(* IEC 61131-3 sources: vscode-twincat-st/src/sample/Errors, 25 files *)

(* ---- C0001.st ---- *)
// C0001: Constant '{constant}' too large for type '{name}'
FUNCTION_BLOCK C0001

    VAR

        // Signed Integer Types
        _int1:                  INT             := INT#2#10000000_00000000;
        _int2:                  INT             := INT#16#8000;

        // Unsigned Integer Types
        _uint1:                 UINT            := UINT#-1;
        _Uint2:                 UINT            := 18446744073709551616;

        // Floating Point Types
        _real:                  REAL            := REAL#3.402824E+38;
        _lreal:                 LREAL           := LREAL#1.7976931348623159e+308;
        _lreal2:                LREAL           := 1.7976931348623159e+308;

        // Time-Related Types
        time_over1:             TIME            := TIME#1M61S;
        time_over2:             TIME            := TIME#49D17H2M47S296MS;

        date_under:             DATE            := DATE#1969-12-31;
		date_over:              DATE            := DATE#2106-02-08;
        date_invalid:           DATE            := D#1970-01-40;

        date_and_time_under:    DATE_AND_TIME   := DATE_AND_TIME#1969-12-31-23:59:59;
        date_and_time_over:     DATE_AND_TIME   := DATE_AND_TIME#2106-02-07-06:28:16;
        date_and_time_invalid:  DATE_AND_TIME   := DATE_AND_TIME#1970-01-40-00:00:00;

        time_of_day_over:       TIME_OF_DAY     := TIME_OF_DAY#24:00:00.000;
        time_of_day_invalid:    TIME_OF_DAY     := TIME_OF_DAY#23:00:72.000;

        l_time_over1:           LTIME           := LTIME#1M61S;
        l_time_over2:           LTIME           := LTIME#213503D23H34M33S709MS551US616NS;

        l_date_under:           LDATE           := LDATE#1969-12-31;
		l_date_over:            LDATE           := LDATE#2554-07-22;

        l_date_and_time_under:  LDATE_AND_TIME  := LDATE_AND_TIME#1969-12-31-23:59:59;
        l_date_and_time_over:   LDATE_AND_TIME  := LDATE_AND_TIME#2554-7-21-23:34:33.709551616;

        l_time_of_day_over:     LTIME_OF_DAY    := LTIME_OF_DAY#24:00:00.000;
    END_VAR
END_FUNCTION_BLOCK

(* ---- C0018.st ---- *)
// C0018 '{name}' is no valid assignment target
FUNCTION_BLOCK C0018

    VAR CONSTANT
        _a: INT;
    END_VAR

    PROPERTY A : INT
        GET
            //
        END_GET
    END_PROPERTY

    METHOD B
        //
    END_METHOD

    _a  := 1;
    A   := 1;
    B   := 1;
END_FUNCTION_BLOCK

(* ---- C0032_DUTs.st ---- *)
// C0032: Cannot convert type '{type}' to type '{type}'

TYPE U_C0032 :
UNION
    A: USINT := 1024;
END_UNION
END_TYPE

TYPE ST_C0032 :
STRUCT
    A: USINT := 1024;
END_STRUCT
END_TYPE

TYPE E_C0032_Default :
(
    A
);
END_TYPE

TYPE E_C0032_USINT :
(
    A := 1024
) USINT;
END_TYPE

TYPE C0032_InnerAlias : E_C0032_USINT;
END_TYPE

TYPE C0032_OuterAlias : C0032_InnerAlias;
END_TYPE

FUNCTION_BLOCK C0032_DUTs

    VAR
        _enum_default:      E_C0032_Default     := 32768;
        _enum_usint:        E_C0032_USINT       := 256;
        _alias:             C0032_OuterAlias    := 256;
        _assign_from_x_1:   USINT               := E_C0032_Default.A;
        _assign_from_x_2:   BOOL;
    END_VAR

    _enum_default       := 32768;
    _enum_usint         := 256;
    _alias              := 256;
    _assign_from_x_1    := E_C0032_Default.A;
    _assign_from_x_1    := _enum_default;
    _assign_from_x_2    := _alias;
END_FUNCTION_BLOCK

(* ---- C0032_Literals.st ---- *)
// C0032: Cannot convert type '{type}' to type '{type}'

FUNCTION_BLOCK C0032_Literals

    VAR

        _a:         BOOL        := 2;
        _subrange:  INT(1..1)   := 2;
    END_VAR

    _a          := 2;
    _subrange   := 2;
END_FUNCTION_BLOCK

(* ---- C0032_Variables.st ---- *)
// C0032: Cannot convert type '{type}' to type '{type}'
// https://infosys.beckhoff.com/english.php?content=../content/1033/tf5100_tc3_nc_i/4188351883.html&id=
FUNCTION_BLOCK C0032_Variables

    VAR
        _bool:  BOOL;
        _byte:  BYTE;
    END_VAR

    _bool := _byte;     // Byte
    _bool := -_byte;    // INT
    _bool := -BYTE#1;   // SINT
END_FUNCTION_BLOCK

(* ---- C0035.st ---- *)
// C0035: Program name, function or function block instance expected instead of '{name}'
FUNCTION_BLOCK FB_C0035

    VAR
        _a: INT;
    END_VAR

    PROPERTY A : INT
        GET
            //
        END_GET
    END_PROPERTY

    METHOD M_A : INT
        //
    END_METHOD

    _a();
    _a := _a();
    E_C0035.a();

    _a := A();
    A();
END_FUNCTION_BLOCK

TYPE E_C0035 :
(
    a
);
END_TYPE

(* ---- C0036.st ---- *)
// C0036: Cannot call object of type '{name}'
FUNCTION_BLOCK FB_C0036
    GVL_C0036();
    E_C0036();
    ST_C0036();
    U_C0036();
END_FUNCTION_BLOCK

VAR_GLOBAL GVL_C0036
    //
END_VAR

TYPE E_C0036 :
(
    dummy
);
END_TYPE

TYPE ST_C0036 :
STRUCT
    //
END_STRUCT
END_TYPE

TYPE U_C0036 :
UNION
    //
END_UNION
END_TYPE

(* ---- C0037.st ---- *)
// C0037: '{name}' is no input of '{name}'

FUNCTION_BLOCK FB_C0037_2

    VAR_OUTPUT
        b: INT;
    END_VAR
END_FUNCTION_BLOCK

FUNCTION_BLOCK FB_C0037

    VAR
        _a: FB_C0037_2;
    END_VAR

    _a.b := 1;
END_FUNCTION_BLOCK

(* ---- C0046.st ---- *)
// C0046: Identifier '{id}' not defined
FUNCTION_BLOCK FB_C0046
    _a := 1;
    THIS^._a();
    _a := THIS^._a();
END_FUNCTION_BLOCK

(* ---- C0047.st ---- *)
// C0047: Cannot apply indexing with [] to an expression of type '{type}'
FUNCTION_BLOCK FB_C0047

    VAR
        _a: INT;
        _b: POINTER TO INT;
    END_VAR

    _a := _a[0];
    _a := _b^[0];
    GVL_C0047[0];
END_FUNCTION_BLOCK

VAR_GLOBAL GVL_C0047
    //
END_VAR

(* ---- C0064.st ---- *)
// C0064: Dereference requires a pointer
FUNCTION_BLOCK FB_C0064

    VAR
        _a:   INT;
        _b:   POINTER TO POINTER TO INT;
    END_VAR

    _a := _a^;
    _a := _b^^^;
    GVL_C0064^;
END_FUNCTION_BLOCK

VAR_GLOBAL GVL_C0064
    //
END_VAR

(* ---- C0066.st ---- *)
// C0066: Cannot compare type '{name}' with type '{name}'
FUNCTION_BLOCK FB_C0066

    VAR
        _a:     INT;
        _b:     TIME;
        _c:     BOOL;
    END_VAR

    _c := _a > _b;
END_FUNCTION_BLOCK

(* ---- C0074.st ---- *)
// C0074: Unexpected array initialisation
FUNCTION_BLOCK FB_C0074

    VAR
       _a: ARRAY [0..1] OF INT;
    END_VAR

    _a := [0, 1];
END_FUNCTION_BLOCK

(* ---- C0077.st ---- *)
// C0077: Unknown type: '{type}'
FUNCTION_BLOCK FB_C0077

    VAR
        _a: UnknownType;
    END_VAR
END_FUNCTION_BLOCK

(* ---- C0080.st ---- *)
// C0080: Function block '{name}' must be instantiated to be accessed
FUNCTION_BLOCK FB_C0080
    FB_C0080();
END_FUNCTION_BLOCK

(* ---- C0140.st ---- *)
// C0140: Reference assign is only allowed to variables of reference type
FUNCTION_BLOCK FB_C0140

    VAR
        _a: INT;
        _b: INT REF= _a;
    END_VAR

    _b REF= _a;
END_FUNCTION_BLOCK

(* ---- C0142.st ---- *)
// C0142: A local variable named '{name}' is already defined in '{scope}'
FUNCTION_BLOCK C0142

    VAR
        A: INT;
        A: INT;
    END_VAR

    PROPERTY A : INT
        GET
            //
        END_GET
    END_PROPERTY
END_FUNCTION_BLOCK

(* ---- C0143.st ---- *)
// C0143: The property '{name}' cannot be used in this context because it lacks the get accessor
FUNCTION_BLOCK C0143

    VAR
        _a: INT;
        _b: C0143_B;
    END_VAR

    PROPERTY A : C0143_B
        SET
            //
        END_SET
    END_PROPERTY

    _a := A.B;
    A.B := _a;
    _b := A;
END_FUNCTION_BLOCK

FUNCTION_BLOCK C0143_B

    PROPERTY B : INT
        GET
            //
        END_GET
        SET
            //
        END_SET
    END_PROPERTY
END_FUNCTION_BLOCK

(* ---- C0177.st ---- *)
// C0177: '{name}' is of type {name} and cannot be instantiated
FUNCTION_BLOCK C0177

    VAR
        _a: PRG_C0177;
        _b: GVL_C0177;
        _c: F_C0177;
    END_VAR
END_FUNCTION_BLOCK

PROGRAM PRG_C0177
    //
END_PROGRAM

VAR_GLOBAL GVL_C0177
    //
END_VAR

FUNCTION F_C0177
    //
END_FUNCTION

(* ---- C0185.st ---- *)
// C0185: It is not possible to perform component access '.', index access '[]' or call '()' on result of function call. Assign result to help variable first.
FUNCTION_BLOCK C0185

    VAR
        _a: INT;
    END_VAR

    PROPERTY A : C0185
        GET
            //
        END_GET
    END_PROPERTY

    PROPERTY B : ARRAY [0..1] OF C0185
        GET
            //
        END_GET
    END_PROPERTY

    METHOD M_A : C0185
        //
    END_METHOD

    METHOD M_B : ARRAY [0..1] OF C0185
        //
    END_METHOD

    // Component access
    M_A().A;

    // Index access
    M_B()[0];

    // Call
    M_A()();
END_FUNCTION_BLOCK

(* ---- C0261.st ---- *)
// C0261: A reference type is not allowed as base type of an array, pointer, or reference
FUNCTION_BLOCK FB_C0261

    VAR
        _a: ARRAY [1..2] OF REFERENCE TO INT;
        _b: POINTER TO REFERENCE TO INT;
        _c: REFERENCE TO REFERENCE TO INT;
    END_VAR
END_FUNCTION_BLOCK

(* ---- M0001.st ---- *)
// M0001: The subrange parameters are not within the valid range
FUNCTION_BLOCK M0001

    VAR
        _a: BYTE(-4095..4095);
    END_VAR
END_FUNCTION_BLOCK

(* ---- M0002.st ---- *)
// M0002: The '{name}' operator is not defined for the types '{name}' and '{name}'
FUNCTION_BLOCK M0002

    VAR
        _bool: BOOL;
    END_VAR

    _bool := _bool + _bool;
END_FUNCTION_BLOCK

(* ---- M0003.st ---- *)
// M0003: The unary operator '{name}' is not defined for type '{name}'
FUNCTION_BLOCK M0003

    VAR
        _a: BOOL;
    END_VAR

    _a := -_a;
END_FUNCTION_BLOCK

(* ---- SA0027.st ---- *)
// SA0027: Object name '{name}' already used in this application
FUNCTION_BLOCK SA0027
    //
END_FUNCTION_BLOCK

FUNCTION_BLOCK SA0027
    //
END_FUNCTION_BLOCK

FUNCTION SA0027
    //
END_FUNCTION
